// Mitsubishi GX Works2 project: test   PLC: FX3U/FX3UC

PROGRAM MAIN
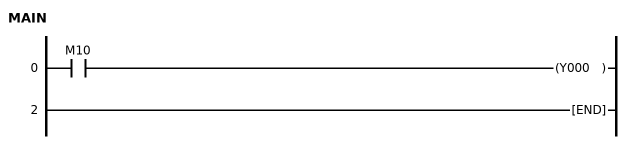
0     LD      M10
      OUT     Y000
2     END
END_PROGRAM
